FUNCTION_BLOCK TcContinuousAxisCommand IMPLEMENTS itfContinuousAxisCommand
VAR_INPUT
END_VAR
VAR_OUTPUT
END_VAR
VAR
END_VAR

{warning 'add method implementation '}
METHOD Abort : MC_Error
END_METHOD

{warning 'add property implementation'}
PROPERTY Active : BOOL
GET
END_GET
END_PROPERTY

{warning 'add property implementation'}
PROPERTY Busy : BOOL
GET
END_GET
END_PROPERTY

{warning 'add property implementation'}
PROPERTY Command : MC_COMMAND_REF
GET
END_GET
END_PROPERTY

{warning 'add property implementation'}
PROPERTY CommandAborted : BOOL
GET
END_GET
END_PROPERTY

{warning 'add property implementation'}
PROPERTY Done : BOOL
GET
END_GET
END_PROPERTY

{warning 'add property implementation'}
PROPERTY Error : BOOL
GET
END_GET
END_PROPERTY

{warning 'add property implementation'}
PROPERTY ErrorId : MC_Error
GET
END_GET
END_PROPERTY

{warning 'add property implementation'}
PROPERTY InVelocity : BOOL
GET
END_GET
END_PROPERTY

{warning 'add method implementation '}
METHOD Update 		: MC_Error
VAR_INPUT
	Position		: REAL;
	Velocity		: REAL;
	EndVelocity		: REAL;
	Acceleration	: REAL;
	Deceleration	: REAL;
	Jerk			: REAL;
END_VAR
END_METHOD

{warning 'add method implementation '}
METHOD Wait 		: MC_Error (* This method only makes sense in the IEC 61499 environment*)
VAR_INPUT
	Timeout			: TIME;
	AbortOnTimeout	: BOOL;
END_VAR
END_METHOD

END_FUNCTION_BLOCK

(* stored: Version 1.1.0.1, ProductVersion 3.1.4024.11
   POU TcContinuousAxisCommand: Id {4161ef74-8cae-4032-9910-f294541a2dec}, SpecialFunc None
   Method Abort: Id {eb9c2030-8593-410b-9f4d-03e78bde1e4d}
   Property Active: Id {ea546285-08b8-49da-87f4-a0a567956075}
   Get Get: Id {ae7ea0d0-59ab-4174-a5e5-71e38e1237f3}
   Property Busy: Id {a282a2df-6993-4e50-9a95-186563112c04}
   Get Get: Id {a41b6987-2289-4b55-9f88-c4032e9b28d4}
   Property Command: Id {1ad29e7c-7398-4c58-adf2-c6934d2731e0}
   Get Get: Id {b2dcc134-3311-4d35-b28c-d22d13f1459c}
   Property CommandAborted: Id {a4f5f460-0bdf-4b3d-8efb-860ebad75552}
   Get Get: Id {3a0f4361-cc16-454d-9327-14e479dca79a}
   Property Done: Id {2b25e5f4-12be-4e3d-a913-b210e3cf2e8a}
   Get Get: Id {b9316619-08ab-4e4a-859b-c02be6822395}
   Property Error: Id {08e4f02c-d77f-4a13-986d-ddacb35c0c2b}
   Get Get: Id {57035b37-5920-430f-bcd4-cd69c1e9cef0}
   Property ErrorId: Id {11c92b9d-f0af-4b75-95d3-1edf3a844d89}
   Get Get: Id {c8a044ff-5c73-477c-91c2-6fc3315e722e}
   Property InVelocity: Id {4af934e6-9d23-46ea-8ff6-1d962c96a6ce}
   Get Get: Id {5c3040ff-6574-407f-b2a5-c575aa6ed355}
   Method Update: Id {2b264c6e-470b-41f7-a1f5-2b2f858d4b99}
   Method Wait: Id {b22357b1-5ebb-4019-977e-820965915fdd} *)
